TYPE ST_MotionOptions :
STRUCT
  eBufferMode   : Tc2_MC2.MC_BufferMode;

END_STRUCT
END_TYPE

(* stored: Version 1.1.0.1, ProductVersion 3.1.4024.12
   DUT ST_MotionOptions: Id {531e3734-24fc-44ad-b289-ab0c650a3e58} *)
